SET P022 P006
SFTON3D P022
SMOVL C00031 BC00031 V=166.7  +MOVJ EC00031
MOVL C00032 BC00032 V=1000.0  +MOVJ EC00032 VJ=100.00
'EndPath S4094
MOVJ C00033 BC00033 VJ=100.00  +MOVJ EC00033 VJ=100.00
'Path S4205
SFTOF3D
MOVJ C00034 BC00034 VJ=100.00  +MOVJ EC00034 VJ=100.00
MOVL C00035 BC00035 V=666.7  +MOVJ EC00035 VJ=100.00
SMOVL C00036 BC00036 V=166.7  +MOVJ EC00036
SREFP 3 C00037 BC00037  +REFP EC00037
CALL JOB:SEARCH-R1-S13D
SET P050 P006
SFTON3D P050
SMOVL C00038 BC00038 V=166.7  +MOVJ EC00038
SREFP 3 C00039 BC00039  +REFP EC00039
CALL JOB:SEARCH-R1-S13D
SET P050 P006
SFTON3D P050
SMOVL C00040 BC00040 V=166.7  +MOVJ EC00040
SMOVL C00041 BC00041 V=250.0  +MOVJ EC00041
SMOVL C00042 BC00042 V=166.7  +MOVJ EC00042
SREFP 3 C00043 BC00043  +REFP EC00043
CALL JOB:SEARCH-R1-S13D
SET P050 P006
SFTON3D P050
SMOVL C00044 BC00044 V=250.0  +MOVJ EC00044
'EndPath S4205
'Path S4206
SFTOF3D
MOVL C00045 BC00045 V=1000.0  +MOVJ EC00045 VJ=100.00
SMOVL C00046 BC00046 V=166.7  +MOVJ EC00046
SREFP 3 C00047 BC00047  +REFP EC00047
CALL JOB:SEARCH-R1-S13D
SET P051 P006
SFTON3D P051
SMOVL C00048 BC00048 V=166.7  +MOVJ EC00048
SREFP 3 C00049 BC00049  +REFP EC00049
CALL JOB:SEARCH-R1-S13D
SET P051 P006
SFTON3D P051
SMOVL C00050 BC00050 V=166.7  +MOVJ EC00050
SMOVL C00051 BC00051 V=250.0  +MOVJ EC00051
SREFP 3 C00052 BC00052  +REFP EC00052
CALL JOB:SEARCH-R1-S13D
SET P051 P006
SFTON3D P051
SMOVL C00053 BC00053 V=250.0  +MOVJ EC00053
MOVL C00054 BC00054 V=1000.0  +MOVJ EC00054 VJ=100.00
'EndPath S4206
MOVJ C00055 BC00055 VJ=100.00  +MOVJ EC00055 VJ=100.00
'Path S4207
SFTOF3D
MOVJ C00056 BC00056 VJ=100.00  +MOVJ EC00056 VJ=100.00
MOVL C00057 BC00057 V=666.7  +MOVJ EC00057 VJ=100.00
SMOVL C00058 BC00058 V=166.7  +MOVJ EC00058
SREFP 3 C00059 BC00059  +REFP EC00059
CALL JOB:SEARCH-R1-S13D
SET P054 P006
SFTON3D P054
SMOVL C00060 BC00060 V=250.0  +MOVJ EC00060
SMOVL C00061 BC00061 V=233.3  +MOVJ EC00061
SMOVL C00062 BC00062 V=166.7  +MOVJ EC00062
SREFP 3 C00063 BC00063  +REFP EC00063
CALL JOB:SEARCH-R1-S13D
SET P054 P006
SFTON3D P054
SMOVL C00064 BC00064 V=166.7  +MOVJ EC00064
SMOVL C00065 BC00065 V=416.7  +MOVJ EC00065
SMOVL C00066 BC00066 V=250.0  +MOVJ EC00066
SREFP 3 C00067 BC00067  +REFP EC00067
CALL JOB:SEARCH-R1-S13D
SET P054 P006
SFTON3D P054
SMOVL C00068 BC00068 V=250.0  +MOVJ EC00068
MOVL C00069 BC00069 V=1000.0  +MOVJ EC00069 VJ=100.00
'EndPath S4207
'Path S4095
SFTOF3D
MOVJ C00070 BC00070 VJ=100.00  +MOVJ EC00070 VJ=100.00
MOVJ C00071 BC00071 VJ=100.00  +MOVJ EC00071 VJ=100.00
SMOVL C00072 BC00072 V=200.0  +MOVJ EC00072
SREFP 3 C00073 BC00073  +REFP EC00073
CALL JOB:SEARCH-R1-S13D
SET P089 P006
SFTON3D P089
SMOVL C00074 BC00074 V=166.7  +MOVJ EC00074
SMOVL C00075 BC00075 V=166.7  +MOVJ EC00075
SREFP 3 C00076 BC00076  +REFP EC00076
CALL JOB:SEARCH-R1-S13D
SET P089 P006
SFTON3D P089
SMOVL C00077 BC00077 V=166.7  +MOVJ EC00077
SMOVL C00078 BC00078 V=166.7  +MOVJ EC00078
SREFP 3 C00079 BC00079  +REFP EC00079
CALL JOB:SEARCH-R1-S13D
SET P089 P006
SFTON3D P089
SMOVL C00080 BC00080 V=166.7  +MOVJ EC00080
SMOVL C00081 BC00081 V=1000.0  +MOVJ EC00081
SFTOF3D
MOVJ C00082 BC00082 VJ=100.00  +MOVJ EC00082 VJ=100.00
MOVL C00083 BC00083 V=666.7  +MOVJ EC00083 VJ=100.00
SMOVL C00084 BC00084 V=166.7  +MOVJ EC00084
SREFP 3 C00085 BC00085  +REFP EC00085
CALL JOB:SEARCH-R1-S13D
SET P034 P006
SFTON3D P034
SMOVL C00086 BC00086 V=250.0  +MOVJ EC00086
SMOVL C00087 BC00087 V=233.3  +MOVJ EC00087
SMOVL C00088 BC00088 V=166.7  +MOVJ EC00088
SREFP 3 C00089 BC00089  +REFP EC00089
CALL JOB:SEARCH-R1-S13D
SET P034 P006
SFTON3D P034
SMOVL C00090 BC00090 V=166.7  +MOVJ EC00090
SMOVL C00091 BC00091 V=166.7  +MOVJ EC00091
SREFP 3 C00092 BC00092  +REFP EC00092
CALL JOB:SEARCH-R1-S13D
SET P034 P006
SFTON3D P034
SMOVL C00093 BC00093 V=166.7  +MOVJ EC00093
MOVJ C00094 BC00094 VJ=50.00  +MOVJ EC00094 VJ=30.00
'EndPath S4095
'Path S4096
SFTOF3D
MOVJ C00095 BC00095 VJ=50.00  +MOVJ EC00095 VJ=30.00
MOVJ C00096 BC00096 VJ=50.00  +MOVJ EC00096 VJ=30.00
MOVJ C00097 BC00097 VJ=50.00  +MOVJ EC00097 VJ=30.00
SMOVL C00098 BC00098 V=166.7  +MOVJ EC00098
SREFP 3 C00099 BC00099  +REFP EC00099
CALL JOB:SEARCH-R1-S13D
SET P061 P006
SFTON3D P061
SMOVL C00100 BC00100 V=166.7  +MOVJ EC00100
SREFP 3 C00101 BC00101  +REFP EC00101
CALL JOB:SEARCH-R1-S13D
SET P061 P006
SFTON3D P061
SMOVL C00102 BC00102 V=166.7  +MOVJ EC00102
SFTOF3D
SMOVL C00103 BC00103 V=666.7  +MOVJ EC00103
SMOVL C00104 BC00104 V=166.7  +MOVJ EC00104
SREFP 3 C00105 BC00105  +REFP EC00105
CALL JOB:SEARCH-R1-S13D
SET P062 P006
SFTON3D P062
SMOVL C00106 BC00106 V=166.7  +MOVJ EC00106
SREFP 3 C00107 BC00107  +REFP EC00107
CALL JOB:SEARCH-R1-S13D
SET P062 P006
SFTON3D P062
SMOVL C00108 BC00108 V=250.0  +MOVJ EC00108
SFTOF3D
SMOVL C00109 BC00109 V=500.0  +MOVJ EC00109
SMOVL C00110 BC00110 V=166.7  +MOVJ EC00110
SREFP 3 C00111 BC00111  +REFP EC00111
CALL JOB:SEARCH-R1-S13D
SET P063 P006
SFTON3D P063
SMOVL C00112 BC00112 V=166.7  +MOVJ EC00112
SREFP 3 C00113 BC00113  +REFP EC00113
CALL JOB:SEARCH-R1-S13D
SET P063 P006
SFTON3D P063
SMOVL C00114 BC00114 V=166.7  +MOVJ EC00114
SFTOF3D
SMOVL C00115 BC00115 V=1000.0  +MOVJ EC00115
MOVJ C00116 BC00116 VJ=100.00  +MOVJ EC00116 VJ=30.00
MOVJ C00117 BC00117 VJ=50.00  +MOVJ EC00117 VJ=30.00
MOVJ C00118 BC00118 VJ=100.00  +MOVJ EC00118 VJ=100.00
MOVL C00119 BC00119 V=666.7  +MOVJ EC00119 VJ=100.00
SMOVL C00120 BC00120 V=166.7  +MOVJ EC00120
SREFP 3 C00121 BC00121  +REFP EC00121
CALL JOB:SEARCH-R1-S13D
SET P023 P006
SFTON3D P023
SMOVL C00122 BC00122 V=166.7  +MOVJ EC00122
SMOVL C00123 BC00123 V=333.3  +MOVJ EC00123
SMOVL C00124 BC00124 V=166.7  +MOVJ EC00124
SREFP 3 C00125 BC00125  +REFP EC00125
CALL JOB:SEARCH-R1-S13D
SET P023 P006
SFTON3D P023
SMOVL C00126 BC00126 V=166.7  +MOVJ EC00126
SMOVL C00127 BC00127 V=166.7  +MOVJ EC00127
SREFP 3 C00128 BC00128  +REFP EC00128
CALL JOB:SEARCH-R1-S13D
SET P023 P006
SFTON3D P023
SMOVL C00129 BC00129 V=166.7  +MOVJ EC00129
MOVL C00130 BC00130 V=1000.0  +MOVJ EC00130 VJ=100.00
'EndPath S4096
MOVJ C00131 BC00131 VJ=100.00  +MOVJ EC00131 VJ=100.00
'Path S4097
SFTOF3D
MOVJ C00132 BC00132 VJ=100.00  +MOVJ EC00132 VJ=100.00
MOVL C00133 BC00133 V=666.7  +MOVJ EC00133 VJ=100.00
SMOVL C00134 BC00134 V=166.7  +MOVJ EC00134
SREFP 3 C00135 BC00135  +REFP EC00135
CALL JOB:SEARCH-R1-S13D
SET P024 P006
SFTON3D P024
SMOVL C00136 BC00136 V=166.7  +MOVJ EC00136
SREFP 3 C00137 BC00137  +REFP EC00137
CALL JOB:SEARCH-R1-S13D
SET P024 P006
SFTON3D P024
SMOVL C00138 BC00138 V=166.7  +MOVJ EC00138
SMOVL C00139 BC00139 V=166.7  +MOVJ EC00139
SREFP 3 C00140 BC00140  +REFP EC00140
CALL JOB:SEARCH-R1-S13D
SET P024 P006
SFTON3D P024
SMOVL C00141 BC00141 V=166.7  +MOVJ EC00141
MOVL C00142 BC00142 V=1000.0  +MOVJ EC00142 VJ=100.00
'EndPath S4097
'Path S4098
SFTOF3D
MOVJ C00143 BC00143 VJ=100.00  +MOVJ EC00143 VJ=100.00
MOVL C00144 BC00144 V=666.7  +MOVJ EC00144 VJ=100.00
SMOVL C00145 BC00145 V=166.7  +MOVJ EC00145
SREFP 3 C00146 BC00146  +REFP EC00146
CALL JOB:SEARCH-R1-S13D
SET P035 P006
SFTON3D P035
SMOVL C00147 BC00147 V=166.7  +MOVJ EC00147
SREFP 3 C00148 BC00148  +REFP EC00148
CALL JOB:SEARCH-R1-S13D
SET P035 P006
SFTON3D P035
SMOVL C00149 BC00149 V=166.7  +MOVJ EC00149
SMOVL C00150 BC00150 V=166.7  +MOVJ EC00150
SMOVL C00151 BC00151 V=166.7  +MOVJ EC00151
SREFP 3 C00152 BC00152  +REFP EC00152
CALL JOB:SEARCH-R1-S13D
SET P035 P006
SFTON3D P035
SMOVL C00153 BC00153 V=166.7  +MOVJ EC00153
MOVL C00154 BC00154 V=1000.0  +MOVJ EC00154 VJ=100.00
'EndPath S4098
'Path S4099
SFTOF3D
MOVJ C00155 BC00155 VJ=100.00  +MOVJ EC00155 VJ=100.00
MOVL C00156 BC00156 V=666.7  +MOVJ EC00156 VJ=100.00
SMOVL C00157 BC00157 V=166.7  +MOVJ EC00157
SREFP 3 C00158 BC00158  +REFP EC00158
CALL JOB:SEARCH-R1-S13D
SET P029 P006
SFTON3D P029
SMOVL C00159 BC00159 V=166.7  +MOVJ EC00159
SREFP 3 C00160 BC00160  +REFP EC00160
CALL JOB:SEARCH-R1-S13D
SET P029 P006
SFTON3D P029
SMOVL C00161 BC00161 V=166.7  +MOVJ EC00161
SMOVL C00162 BC00162 V=250.0  +MOVJ EC00162
SMOVL C00163 BC00163 V=166.7  +MOVJ EC00163
SREFP 3 C00164 BC00164  +REFP EC00164
CALL JOB:SEARCH-R1-S13D
SET P029 P006
SFTON3D P029
SMOVL C00165 BC00165 V=166.7  +MOVJ EC00165
'EndPath S4099
'Path S4855
SFTOF3D
MOVL C00166 BC00166 V=666.7  +MOVJ EC00166 VJ=100.00
SMOVL C00167 BC00167 V=166.7  +MOVJ EC00167
SREFP 3 C00168 BC00168  +REFP EC00168
CALL JOB:SEARCH-R1-S13D
SET P071 P006
SFTON3D P071
SMOVL C00169 BC00169 V=166.7  +MOVJ EC00169
SREFP 3 C00170 BC00170  +REFP EC00170
CALL JOB:SEARCH-R1-S13D
SET P071 P006
SFTON3D P071
SMOVL C00171 BC00171 V=166.7  +MOVJ EC00171
SMOVL C00172 BC00172 V=166.7  +MOVJ EC00172
SREFP 3 C00173 BC00173  +REFP EC00173
CALL JOB:SEARCH-R1-S13D
SET P071 P006
SFTON3D P071
SMOVL C00174 BC00174 V=166.7  +MOVJ EC00174
MOVL C00175 BC00175 V=1000.0  +MOVJ EC00175 VJ=100.00
'EndPath S4855
'Path S4856
SFTOF3D
MOVJ C00176 BC00176 VJ=100.00  +MOVJ EC00176 VJ=100.00
MOVL C00177 BC00177 V=666.7  +MOVJ EC00177 VJ=100.00
SMOVL C00178 BC00178 V=166.7  +MOVJ EC00178
SREFP 3 C00179 BC00179  +REFP EC00179
CALL JOB:SEARCH-R1-S13D
SET P072 P006
SFTON3D P072
SMOVL C00180 BC00180 V=166.7  +MOVJ EC00180
SREFP 3 C00181 BC00181  +REFP EC00181
CALL JOB:SEARCH-R1-S13D
SET P072 P006
SFTON3D P072
SMOVL C00182 BC00182 V=166.7  +MOVJ EC00182
MOVL C00183 BC00183 V=1000.0  +MOVJ EC00183 VJ=100.00
'EndPath S4856
MOVJ C00184 BC00184 VJ=100.00  +MOVJ EC00184 VJ=100.00
'Path S4857
SFTOF3D
MOVJ C00185 BC00185 VJ=100.00  +MOVJ EC00185 VJ=100.00
MOVL C00186 BC00186 V=666.7  +MOVJ EC00186 VJ=100.00
SMOVL C00187 BC00187 V=166.7  +MOVJ EC00187
SREFP 3 C00188 BC00188  +REFP EC00188
CALL JOB:SEARCH-R1-S13D
SET P073 P006
SFTON3D P073
SMOVL C00189 BC00189 V=166.7  +MOVJ EC00189
SMOVL C00190 BC00190 V=166.7  +MOVJ EC00190
SREFP 3 C00191 BC00191  +REFP EC00191
CALL JOB:SEARCH-R1-S13D
SET P073 P006
SFTON3D P073
SMOVL C00192 BC00192 V=166.7  +MOVJ EC00192
SMOVL C00193 BC00193 V=166.7  +MOVJ EC00193
SREFP 3 C00194 BC00194  +REFP EC00194
CALL JOB:SEARCH-R1-S13D
SET P073 P006
SFTON3D P073
SMOVL C00195 BC00195 V=166.7  +MOVJ EC00195
MOVL C00196 BC00196 V=1000.0  +MOVJ EC00196 VJ=100.00
'EndPath S4857
MOVJ C00197 BC00197 VJ=100.00  +MOVJ EC00197 VJ=100.00
'Path S4858
SFTOF3D
MOVJ C00198 BC00198 VJ=100.00  +MOVJ EC00198 VJ=100.00
MOVL C00199 BC00199 V=666.7  +MOVJ EC00199 VJ=100.00
SMOVL C00200 BC00200 V=166.7  +MOVJ EC00200
SREFP 3 C00201 BC00201  +REFP EC00201
CALL JOB:SEARCH-R1-S13D
SET P074 P006
SFTON3D P074
SMOVL C00202 BC00202 V=166.7  +MOVJ EC00202
SREFP 3 C00203 BC00203  +REFP EC00203
CALL JOB:SEARCH-R1-S13D
SET P074 P006
SFTON3D P074
SMOVL C00204 BC00204 V=166.7  +MOVJ EC00204
MOVL C00205 BC00205 V=1000.0  +MOVJ EC00205 VJ=100.00
'EndPath S4858
MOVJ C00206 BC00206 VJ=100.00  +MOVJ EC00206 VJ=100.00
MOVJ C00207 BC00207 VJ=100.00  +MOVJ EC00207 VJ=100.00
'Path S4100
SFTOF3D
MOVJ C00208 BC00208 VJ=100.00  +MOVJ EC00208 VJ=100.00
MOVL C00209 BC00209 V=666.7  +MOVJ EC00209 VJ=100.00
SMOVL C00210 BC00210 V=166.7  +MOVJ EC00210
SREFP 3 C00211 BC00211  +REFP EC00211
CALL JOB:SEARCH-R1-S13D
SET P026 P006
SFTON3D P026
SMOVL C00212 BC00212 V=166.7  +MOVJ EC00212
SREFP 3 C00213 BC00213  +REFP EC00213
CALL JOB:SEARCH-R1-S13D
SET P026 P006
SFTON3D P026
SMOVL C00214 BC00214 V=166.7  +MOVJ EC00214
SMOVL C00215 BC00215 V=666.7  +MOVJ EC00215
SMOVL C00216 BC00216 V=666.7  +MOVJ EC00216
SMOVL C00217 BC00217 V=666.7  +MOVJ EC00217
SMOVL C00218 BC00218 V=166.7  +MOVJ EC00218
SREFP 3 C00219 BC00219  +REFP EC00219
CALL JOB:SEARCH-R1-S13D
SET P026 P006
SFTON3D P026
SMOVL C00220 BC00220 V=250.0  +MOVJ EC00220
SMOVL C00221 BC00221 V=666.7  +MOVJ EC00221
MOVL C00222 BC00222 V=1000.0  +MOVJ EC00222 VJ=100.00
'EndPath S4100
MOVJ C00223 BC00223 VJ=50.00  +MOVJ EC00223 VJ=100.00
'Path S4101
SFTOF3D
MOVJ C00224 BC00224 VJ=50.00  +MOVJ EC00224 VJ=100.00
MOVL C00225 BC00225 V=666.7  +MOVJ EC00225 VJ=100.00
SMOVL C00226 BC00226 V=166.7  +MOVJ EC00226
SREFP 3 C00227 BC00227  +REFP EC00227
CALL JOB:SEARCH-R1-S13D
SET P025 P006
SFTON3D P025
SMOVL C00228 BC00228 V=166.7  +MOVJ EC00228
SREFP 3 C00229 BC00229  +REFP EC00229
CALL JOB:SEARCH-R1-S13D
SET P025 P006
SFTON3D P025
SMOVL C00230 BC00230 V=166.7  +MOVJ EC00230
SMOVL C00231 BC00231 V=333.3  +MOVJ EC00231
SMOVL C00232 BC00232 V=166.7  +MOVJ EC00232
SREFP 3 C00233 BC00233  +REFP EC00233
CALL JOB:SEARCH-R1-S13D
SET P025 P006
SFTON3D P025
SMOVL C00234 BC00234 V=166.7  +MOVJ EC00234
MOVL C00235 BC00235 V=1000.0  +MOVJ EC00235 VJ=100.00
'EndPath S4101
MOVJ C00236 BC00236 VJ=100.00  +MOVJ EC00236 VJ=100.00
'Path S4102
SFTOF3D
MOVJ C00237 BC00237 VJ=100.00  +MOVJ EC00237 VJ=100.00
MOVL C00238 BC00238 V=666.7  +MOVJ EC00238 VJ=100.00
SMOVL C00239 BC00239 V=166.7  +MOVJ EC00239
SREFP 3 C00240 BC00240  +REFP EC00240
CALL JOB:SEARCH-R1-S13D
SET P028 P006
SFTON3D P028
SMOVL C00241 BC00241 V=166.7  +MOVJ EC00241
SREFP 3 C00242 BC00242  +REFP EC00242
CALL JOB:SEARCH-R1-S13D
SET P028 P006
SFTON3D P028
SMOVL C00243 BC00243 V=166.7  +MOVJ EC00243
SMOVL C00244 BC00244 V=333.3  +MOVJ EC00244
SMOVL C00245 BC00245 V=166.7  +MOVJ EC00245
SREFP 3 C00246 BC00246  +REFP EC00246
CALL JOB:SEARCH-R1-S13D
SET P028 P006
SFTON3D P028
SMOVL C00247 BC00247 V=166.7  +MOVJ EC00247
MOVL C00248 BC00248 V=1000.0  +MOVJ EC00248 VJ=100.00
'EndPath S4102
MOVJ C00249 BC00249 VJ=100.00  +MOVJ EC00249 VJ=100.00
'Path S4103
SFTOF3D
MOVJ C00250 BC00250 VJ=100.00  +MOVJ EC00250 VJ=100.00
MOVL C00251 BC00251 V=666.7  +MOVJ EC00251 VJ=100.00
SMOVL C00252 BC00252 V=166.7  +MOVJ EC00252
SREFP 3 C00253 BC00253  +REFP EC00253
CALL JOB:SEARCH-R1-S13D
SET P033 P006
SFTON3D P033
SMOVL C00254 BC00254 V=166.7  +MOVJ EC00254
SMOVL C00255 BC00255 V=166.7  +MOVJ EC00255
SREFP 3 C00256 BC00256  +REFP EC00256
CALL JOB:SEARCH-R1-S13D
SET P033 P006
SFTON3D P033
SMOVL C00257 BC00257 V=166.7  +MOVJ EC00257
SMOVL C00258 BC00258 V=166.7  +MOVJ EC00258
SMOVL C00259 BC00259 V=166.7  +MOVJ EC00259
SREFP 3 C00260 BC00260  +REFP EC00260
CALL JOB:SEARCH-R1-S13D
SET P033 P006
SFTON3D P033
SMOVL C00261 BC00261 V=166.7  +MOVJ EC00261
MOVL C00262 BC00262 V=1000.0  +MOVJ EC00262 VJ=100.00
'EndPath S4103
'Path S4104
SFTOF3D
MOVJ C00263 BC00263 VJ=100.00  +MOVJ EC00263 VJ=100.00
MOVL C00264 BC00264 V=666.7  +MOVJ EC00264 VJ=100.00
SMOVL C00265 BC00265 V=166.7  +MOVJ EC00265
SREFP 3 C00266 BC00266  +REFP EC00266
CALL JOB:SEARCH-R1-S13D
SET P027 P006
SFTON3D P027
SMOVL C00267 BC00267 V=250.0  +MOVJ EC00267
SMOVL C00268 BC00268 V=166.7  +MOVJ EC00268
SREFP 3 C00269 BC00269  +REFP EC00269
CALL JOB:SEARCH-R1-S13D
SET P027 P006
SFTON3D P027
SMOVL C00270 BC00270 V=166.7  +MOVJ EC00270
SMOVL C00271 BC00271 V=166.7  +MOVJ EC00271
SREFP 3 C00272 BC00272  +REFP EC00272
CALL JOB:SEARCH-R1-S13D
SET P027 P006
SFTON3D P027
SMOVL C00273 BC00273 V=166.7  +MOVJ EC00273
MOVL C00274 BC00274 V=1000.0  +MOVJ EC00274 VJ=100.00
'EndPath S4104
MOVJ C00275 BC00275 VJ=100.00  +MOVJ EC00275 VJ=100.00
'Path S4105
SFTOF3D
MOVJ C00276 BC00276 VJ=100.00  +MOVJ EC00276 VJ=100.00
MOVL C00277 BC00277 V=666.7  +MOVJ EC00277 VJ=100.00
SMOVL C00278 BC00278 V=166.7  +MOVJ EC00278
SREFP 3 C00279 BC00279  +REFP EC00279
CALL JOB:SEARCH-R1-S13D
SET P030 P006
SFTON3D P030
SMOVL C00280 BC00280 V=166.7  +MOVJ EC00280
SREFP 3 C00281 BC00281  +REFP EC00281
CALL JOB:SEARCH-R1-S13D
SET P030 P006
SFTON3D P030
SMOVL C00282 BC00282 V=166.7  +MOVJ EC00282
MOVL C00283 BC00283 V=1000.0  +MOVJ EC00283 VJ=100.00
'EndPath S4105
'Path S4106
SFTOF3D
MOVJ C00284 BC00284 VJ=100.00  +MOVJ EC00284 VJ=100.00
MOVL C00285 BC00285 V=666.7  +MOVJ EC00285 VJ=100.00
SMOVL C00286 BC00286 V=166.7  +MOVJ EC00286
SREFP 3 C00287 BC00287  +REFP EC00287
CALL JOB:SEARCH-R1-S13D
SET P031 P006
SFTON3D P031
SMOVL C00288 BC00288 V=166.7  +MOVJ EC00288
SREFP 3 C00289 BC00289  +REFP EC00289
CALL JOB:SEARCH-R1-S13D
SET P031 P006
SFTON3D P031
SMOVL C00290 BC00290 V=166.7  +MOVJ EC00290
MOVL C00291 BC00291 V=1000.0  +MOVJ EC00291 VJ=100.00
'EndPath S4106
MOVJ C00292 BC00292 VJ=100.00  +MOVJ EC00292 VJ=100.00
'Path S4107
SFTOF3D
MOVJ C00293 BC00293 VJ=100.00  +MOVJ EC00293 VJ=100.00
MOVL C00294 BC00294 V=666.7  +MOVJ EC00294 VJ=100.00
SMOVL C00295 BC00295 V=166.7  +MOVJ EC00295
SREFP 3 C00296 BC00296  +REFP EC00296
CALL JOB:SEARCH-R1-S13D
SET P032 P006
SFTON3D P032
SMOVL C00297 BC00297 V=166.7  +MOVJ EC00297
SREFP 3 C00298 BC00298  +REFP EC00298
CALL JOB:SEARCH-R1-S13D
SET P032 P006
SFTON3D P032
SMOVL C00299 BC00299 V=166.7  +MOVJ EC00299
SMOVL C00300 BC00300 V=250.0  +MOVJ EC00300
SMOVL C00301 BC00301 V=166.7  +MOVJ EC00301
SREFP 3 C00302 BC00302  +REFP EC00302
CALL JOB:SEARCH-R1-S13D
SET P032 P006
SFTON3D P032
SMOVL C00303 BC00303 V=166.7  +MOVJ EC00303
MOVL C00304 BC00304 V=1000.0  +MOVJ EC00304 VJ=100.00
'EndPath S4107
'
MOVJ C00305 BC00305 VJ=100.00  +MOVJ EC00305 VJ=100.00
'Path S4208
SFTOF3D
MOVJ C00306 BC00306 VJ=100.00  +MOVJ EC00306 VJ=100.00
MOVL C00307 BC00307 V=666.7  +MOVJ EC00307 VJ=100.00
SMOVL C00308 BC00308 V=166.7  +MOVJ EC00308
SREFP 3 C00309 BC00309  +REFP EC00309
CALL JOB:SEARCH-R1-S13D
SET P052 P006
SFTON3D P052
SMOVL C00310 BC00310 V=166.7  +MOVJ EC00310
SREFP 3 C00311 BC00311  +REFP EC00311
CALL JOB:SEARCH-R1-S13D
SET P052 P006
SFTON3D P052
SMOVL C00312 BC00312 V=166.7  +MOVJ EC00312
SFTOF3D
MOVL C00313 BC00313 V=1000.0  +MOVJ EC00313 VJ=100.00
SMOVL C00314 BC00314 V=500.0  +MOVJ EC00314
SMOVL C00315 BC00315 V=166.7  +MOVJ EC00315
SREFP 3 C00316 BC00316  +REFP EC00316
CALL JOB:SEARCH-R1-S13D
SET P088 P006
SFTON3D P088
SMOVL C00317 BC00317 V=166.7  +MOVJ EC00317
SMOVL C00318 BC00318 V=166.7  +MOVJ EC00318
SMOVL C00319 BC00319 V=166.7  +MOVJ EC00319
SREFP 3 C00320 BC00320  +REFP EC00320
CALL JOB:SEARCH-R1-S13D
SET P088 P006
SFTON3D P088
SMOVL C00321 BC00321 V=333.3  +MOVJ EC00321
SMOVL C00322 BC00322 V=666.7  +MOVJ EC00322
SFTOF3D
'EndPath S4208
MOVJ C00323 BC00323 VJ=100.00  +MOVJ EC00323 VJ=100.00
'Path S4209
SFTOF3D
MOVJ C00324 BC00324 VJ=100.00  +MOVJ EC00324 VJ=100.00
MOVL C00325 BC00325 V=666.7  +MOVJ EC00325 VJ=100.00
SMOVL C00326 BC00326 V=166.7  +MOVJ EC00326
SREFP 3 C00327 BC00327  +REFP EC00327
CALL JOB:SEARCH-R1-S13D
SET P053 P006
SFTON3D P053
SMOVL C00328 BC00328 V=166.7  +MOVJ EC00328
SMOVL C00329 BC00329 V=166.7  +MOVJ EC00329
SREFP 3 C00330 BC00330  +REFP EC00330
CALL JOB:SEARCH-R1-S13D
SET P053 P006
SFTON3D P053
SMOVL C00331 BC00331 V=166.7  +MOVJ EC00331
MOVL C00332 BC00332 V=1000.0  +MOVJ EC00332 VJ=100.00
'EndPath S4209
*BP1
MOVJ C00333 BC00333 VJ=100.00  +MOVJ EC00333 VJ=100.00
'Path W4108
SFTOF3D
SFTON3D P033
MOVJ C00334 BC00334 VJ=100.00  +MOVJ EC00334 VJ=100.00
SMOVL C00335 BC00335 V=666.7  +MOVJ EC00335
SMOVL C00336 BC00336 V=166.7 PL=0  +MOVJ EC00336
MACRO1 MJ#(0) ARGF14
ARCON
SMOVL C00337 BC00337 V=9.2  +MOVJ EC00337
ARCOF
SMOVL C00338 BC00338 V=800.0  +MOVJ EC00338
SMOVL C00339 BC00339 V=1000.0  +MOVJ EC00339
SFTOF3D
'EndPath W4108
'Path W4109
SFTOF3D
MOVJ C00340 BC00340 VJ=100.00  +MOVJ EC00340 VJ=100.00
MOVJ C00341 BC00341 VJ=100.00  +MOVJ EC00341 VJ=100.00
'Path W4110
SFTOF3D
SFTON3D P033
MOVJ C00342 BC00342 VJ=100.00  +MOVJ EC00342 VJ=100.00
SMOVL C00343 BC00343 V=800.0  +MOVJ EC00343
SMOVL C00344 BC00344 V=133.3 PL=0  +MOVJ EC00344
MACRO1 MJ#(0) ARGF9
ARCON
SMOVL C00345 BC00345 V=11.7  +MOVJ EC00345
SMOVL C00346 BC00346 V=11.7  +MOVJ EC00346
SMOVL C00347 BC00347 V=11.7  +MOVJ EC00347
ARCOF
SMOVL C00348 BC00348 V=800.0  +MOVJ EC00348
SMOVL C00349 BC00349 V=1000.0  +MOVJ EC00349
SFTOF3D
'EndPath W4110
MOVJ C00350 BC00350 VJ=100.00  +MOVJ EC00350 VJ=100.00
'9
MOVJ C00351 BC00351 VJ=100.00  +MOVJ EC00351 VJ=100.00
'Path W4111
SFTOF3D
SFTON3D P026
MOVJ C00352 BC00352 VJ=100.00  +MOVJ EC00352 VJ=100.00
SMOVL C00353 BC00353 V=666.7  +MOVJ EC00353
SMOVL C00354 BC00354 V=166.7 PL=0  +MOVJ EC00354
MACRO1 MJ#(0) ARGF14
ARCON
SMOVL C00355 BC00355 V=9.2  +MOVJ EC00355
ARCOF
SMOVL C00356 BC00356 V=800.0  +MOVJ EC00356
SMOVL C00357 BC00357 V=1000.0  +MOVJ EC00357
SFTOF3D
'EndPath W4111
'Path W4112
SFTOF3D
SFTON3D P026
MOVJ C00358 BC00358 VJ=100.00  +MOVJ EC00358 VJ=100.00
SMOVL C00359 BC00359 V=800.0  +MOVJ EC00359
SMOVL C00360 BC00360 V=150.0 PL=0  +MOVJ EC00360
ARCON
SMOVL C00361 BC00361 V=11.7  +MOVJ EC00361
SMOVL C00362 BC00362 V=11.7  +MOVJ EC00362
SMOVL C00363 BC00363 V=11.7  +MOVJ EC00363
ARCOF
SMOVL C00364 BC00364 V=800.0  +MOVJ EC00364
SMOVL C00365 BC00365 V=1000.0  +MOVJ EC00365
SFTOF3D
MOVJ C00366 BC00366 VJ=100.00  +MOVJ EC00366 VJ=100.00
MOVJ C00367 BC00367 VJ=100.00  +MOVJ EC00367 VJ=100.00
'uwaga na podajnik
'Path W4114
SFTOF3D
SFTON3D P026
MOVJ C00368 BC00368 VJ=100.00  +MOVJ EC00368 VJ=100.00
SMOVL C00369 BC00369 V=800.0  +MOVJ EC00369
SMOVL C00370 BC00370 V=150.0 PL=0  +MOVJ EC00370
ARCON
SMOVL C00371 BC00371 V=11.7  +MOVJ EC00371
SMOVL C00372 BC00372 V=11.7  +MOVJ EC00372
ARCOF
SMOVL C00373 BC00373 V=800.0  +MOVJ EC00373
SMOVL C00374 BC00374 V=1000.0  +MOVJ EC00374
SFTOF3D
'EndPath W4114
'brak dostepu offset drutu 1cm
'Path W4115
SFTOF3D
SFTON3D P026
MOVJ C00375 BC00375 VJ=100.00  +MOVJ EC00375 VJ=100.00
SMOVL C00376 BC00376 V=800.0  +MOVJ EC00376
SMOVL C00377 BC00377 V=150.0 PL=0  +MOVJ EC00377
ARCON
SMOVL C00378 BC00378 V=11.7  +MOVJ EC00378
ARCOF
SMOVL C00379 BC00379 V=800.0  +MOVJ EC00379
SMOVL C00380 BC00380 V=1000.0  +MOVJ EC00380
SFTOF3D
'EndPath W4115
MOVJ C00381 BC00381 VJ=100.00  +MOVJ EC00381 VJ=100.00
'10
'11
MOVJ C00382 BC00382 VJ=100.00  +MOVJ EC00382 VJ=100.00
'Path W4118
SFTOF3D
SFTON3D P025
MOVJ C00383 BC00383 VJ=100.00  +MOVJ EC00383 VJ=100.00
SMOVL C00384 BC00384 V=800.0  +MOVJ EC00384
SMOVL C00385 BC00385 V=166.7  +MOVJ EC00385
ARCON
SMOVL C00386 BC00386 V=9.2  +MOVJ EC00386
SMOVL C00387 BC00387 V=9.2  +MOVJ EC00387
SMOVL C00388 BC00388 V=9.2  +MOVJ EC00388
SMOVL C00389 BC00389 V=9.2  +MOVJ EC00389
SMOVL C00390 BC00390 V=9.2  +MOVJ EC00390
ARCOF
SMOVL C00391 BC00391 V=800.0  +MOVJ EC00391
SMOVL C00392 BC00392 V=1000.0  +MOVJ EC00392
SFTOF3D
'EndPath W4118
'brak dostepu offset drutu 1cm
MOVJ C00393 BC00393 VJ=100.00  +MOVJ EC00393 VJ=100.00
'Path W4117
SFTOF3D
SFTON3D P025
MOVJ C00394 BC00394 VJ=100.00  +MOVJ EC00394 VJ=100.00
SMOVL C00395 BC00395 V=800.0  +MOVJ EC00395
SMOVL C00396 BC00396 V=166.7 PL=0  +MOVJ EC00396
ARCON
SMOVL C00397 BC00397 V=10.0  +MOVJ EC00397
ARCOF
SMOVL C00398 BC00398 V=800.0  +MOVJ EC00398
SMOVL C00399 BC00399 V=1000.0  +MOVJ EC00399
SFTOF3D
'EndPath W4117
'12
MOVJ C00400 BC00400 VJ=100.00  +MOVJ EC00400 VJ=100.00
MOVJ C00401 BC00401 VJ=100.00  +MOVJ EC00401 VJ=100.00
'Path W4859
SFTOF3D
SFTON3D P073
MOVJ C00402 BC00402 VJ=100.00  +MOVJ EC00402 VJ=100.00
SMOVL C00403 BC00403 V=800.0  +MOVJ EC00403
SMOVL C00404 BC00404 V=150.0 PL=0  +MOVJ EC00404
ARCON
SMOVL C00405 BC00405 V=8.3  +MOVJ EC00405
SFTON3D P074
SMOVL C00406 BC00406 V=9.2  +MOVJ EC00406
SMOVL C00407 BC00407 V=9.2  +MOVJ EC00407
ARCOF
SMOVL C00408 BC00408 V=800.0  +MOVJ EC00408
SMOVL C00409 BC00409 V=1000.0  +MOVJ EC00409
SFTOF3D
'EndPath W4859
MOVJ C00410 BC00410 VJ=100.00  +MOVJ EC00410 VJ=100.00
MOVJ C00411 BC00411 VJ=100.00  +MOVJ EC00411 VJ=100.00
'Path W4119
SFTOF3D
SFTON3D P034
MOVJ C00412 BC00412 VJ=100.00  +MOVJ EC00412 VJ=100.00
SMOVL C00413 BC00413 V=800.0  +MOVJ EC00413
SMOVL C00414 BC00414 V=150.0 PL=0  +MOVJ EC00414
ARCON
SMOVL C00415 BC00415 V=10.0  +MOVJ EC00415
SMOVL C00416 BC00416 V=10.0  +MOVJ EC00416
SMOVL C00417 BC00417 V=10.0  +MOVJ EC00417
ARCOF
SMOVL C00418 BC00418 V=800.0  +MOVJ EC00418
SMOVL C00419 BC00419 V=1000.0  +MOVJ EC00419
SFTOF3D
'EndPath W4119
'Path W4210
SFTOF3D
SFTON3D P050
MOVJ C00420 BC00420 VJ=100.00  +MOVJ EC00420 VJ=100.00
SMOVL C00421 BC00421 V=800.0  +MOVJ EC00421
SMOVL C00422 BC00422 V=150.0 PL=0  +MOVJ EC00422
ARCON
SMOVL C00423 BC00423 V=11.7  +MOVJ EC00423
ARCOF
SMOVL C00424 BC00424 V=800.0  +MOVJ EC00424
SMOVL C00425 BC00425 V=1000.0  +MOVJ EC00425
SFTOF3D
'EndPath W4210
'Path W4211
SFTOF3D
SFTON3D P034
MOVJ C00426 BC00426 VJ=100.00  +MOVJ EC00426 VJ=100.00
SMOVL C00427 BC00427 V=800.0  +MOVJ EC00427
SMOVL C00428 BC00428 V=166.7 PL=0  +MOVJ EC00428
ARCON
SWVON WEV#(66)
SMOVL C00429 BC00429 V=9.2  +MOVJ EC00429
SMOVL C00430 BC00430 V=9.2  +MOVJ EC00430
SMOVL C00431 BC00431 V=9.2  +MOVJ EC00431
ARCOF
WVOF
SMOVL C00432 BC00432 V=800.0  +MOVJ EC00432
SMOVL C00433 BC00433 V=1000.0  +MOVJ EC00433
MOVJ C00434 BC00434 VJ=30.00  +MOVJ EC00434 VJ=30.00
MOVJ C00435 BC00435 VJ=30.00  +MOVJ EC00435 VJ=30.00
SFTOF3D
MACRO1 MJ#(0) ARGF6
MOVJ C00436 BC00436 VJ=30.00  +MOVJ EC00436 VJ=30.00
SFTON3D P063
SMOVL C00437 BC00437 V=133.3  +MOVJ EC00437
ARCON
SMOVL C00438 BC00438 V=11.7  +MOVJ EC00438
SMOVL C00439 BC00439 V=11.7  +MOVJ EC00439
SMOVL C00440 BC00440 V=11.7  +MOVJ EC00440
SFTON3D P062
SMOVL C00441 BC00441 V=11.7  +MOVJ EC00441
SMOVL C00442 BC00442 V=11.7  +MOVJ EC00442
SFTON3D P061
SMOVL C00443 BC00443 V=11.0  +MOVJ EC00443
SMOVL C00444 BC00444 V=11.0  +MOVJ EC00444
ARCOF
SMOVL C00445 BC00445 V=250.0  +MOVJ EC00445
SFTOF3D
MOVJ C00446 BC00446 VJ=20.00  +MOVJ EC00446 VJ=20.00
MOVJ C00447 BC00447 VJ=20.00  +MOVJ EC00447 VJ=20.00
MOVJ C00448 BC00448 VJ=30.00  +MOVJ EC00448 VJ=30.00
'EndPath W4211
'Path W4210
SFTOF3D
SFTON3D P054
MOVJ C00449 BC00449 VJ=100.00  +MOVJ EC00449 VJ=100.00
SMOVL C00450 BC00450 V=800.0  +MOVJ EC00450
SMOVL C00451 BC00451 V=150.0 PL=0  +MOVJ EC00451
MACRO1 MJ#(0) ARGF14
ARCON
SWVON WEV#(67)
SMOVL C00452 BC00452 V=10.0  +MOVJ EC00452
SMOVL C00453 BC00453 V=10.0  +MOVJ EC00453
ARCOF
SWVOF
SMOVL C00454 BC00454 V=800.0  +MOVJ EC00454
SMOVL C00455 BC00455 V=1000.0  +MOVJ EC00455
SFTOF3D
'EndPath W4210
'Path W4121
SFTOF3D
SFTON3D P028
MOVJ C00456 BC00456 VJ=100.00  +MOVJ EC00456 VJ=100.00
SMOVL C00457 BC00457 V=800.0  +MOVJ EC00457
SMOVL C00458 BC00458 V=150.0 PL=0  +MOVJ EC00458
ARCON
SMOVL C00459 BC00459 V=9.2  +MOVJ EC00459
SMOVL C00460 BC00460 V=9.2  +MOVJ EC00460
SMOVL C00461 BC00461 V=9.2  +MOVJ EC00461
ARCOF
SMOVL C00462 BC00462 V=800.0  +MOVJ EC00462
SMOVL C00463 BC00463 V=1000.0  +MOVJ EC00463
SFTOF3D
'EndPath W4121
'brak dostepu offset 5mm
MOVJ C00464 BC00464 VJ=100.00  +MOVJ EC00464 VJ=100.00
'Path W4122
SFTOF3D
SFTON3D P028
MOVJ C00465 BC00465 VJ=100.00  +MOVJ EC00465 VJ=100.00
SMOVL C00466 BC00466 V=800.0  +MOVJ EC00466
SMOVL C00467 BC00467 V=166.7 PL=0  +MOVJ EC00467
ARCON
SMOVL C00468 BC00468 V=11.7  +MOVJ EC00468
ARCOF
SMOVL C00469 BC00469 V=800.0  +MOVJ EC00469
SMOVL C00470 BC00470 V=1000.0  +MOVJ EC00470
SFTOF3D
'EndPath W4122
MOVJ C00471 BC00471 VJ=100.00  +MOVJ EC00471 VJ=100.00
'13
MOVJ C00472 BC00472 VJ=100.00  +MOVJ EC00472 VJ=100.00
'Path W4123
SFTOF3D
SFTON3D P030
MOVJ C00473 BC00473 VJ=100.00  +MOVJ EC00473 VJ=100.00
SMOVL C00474 BC00474 V=800.0  +MOVJ EC00474
SMOVL C00475 BC00475 V=150.0 PL=0  +MOVJ EC00475
MACRO1 MJ#(0) ARGF9
ARCON
SWVON WEV#(10)
SFTON3D P031
SMOVL C00476 BC00476 V=12.5  +MOVJ EC00476
ARCOF
SWVOF
SMOVL C00477 BC00477 V=800.0  +MOVJ EC00477
SMOVL C00478 BC00478 V=1000.0  +MOVJ EC00478
SFTOF3D
'EndPath W4123
'14
'15-brak
'Path W4212
SFTOF3D
SFTON3D P052
MOVJ C00479 BC00479 VJ=100.00  +MOVJ EC00479 VJ=100.00
SMOVL C00480 BC00480 V=800.0  +MOVJ EC00480
SMOVL C00481 BC00481 V=150.0 PL=0  +MOVJ EC00481
ARCON
SMOVL C00482 BC00482 V=10.8  +MOVJ EC00482
SMOVL C00483 BC00483 V=10.8  +MOVJ EC00483
SMOVL C00484 BC00484 V=10.8  +MOVJ EC00484
ARCOF
SMOVL C00485 BC00485 V=800.0  +MOVJ EC00485
MACRO1 MJ#(0) ARGF6
SMOVL C00486 BC00486 V=333.3  +MOVJ EC00486
SFTOF3D
'DODAC SHIFT
SFTON3D P088
SMOVL C00487 BC00487 V=133.3  +MOVJ EC00487
ARCON
SMOVL C00488 BC00488 V=10.8  +MOVJ EC00488
ARCOF
SMOVL C00489 BC00489 V=250.0  +MOVJ EC00489
SMOVL C00490 BC00490 V=1000.0  +MOVJ EC00490
SFTOF3D
'EndPath W4212
'16
'Path W4213
SFTOF3D
SFTON3D P053
MOVJ C00491 BC00491 VJ=100.00  +MOVJ EC00491 VJ=100.00
SMOVL C00492 BC00492 V=800.0  +MOVJ EC00492
SMOVL C00493 BC00493 V=150.0 PL=0  +MOVJ EC00493
MACRO1 MJ#(0) ARGF9
ARCON
SMOVL C00494 BC00494 V=10.8  +MOVJ EC00494
SMOVL C00495 BC00495 V=10.8  +MOVJ EC00495
SMOVL C00496 BC00496 V=10.8  +MOVJ EC00496
ARCOF
SMOVL C00497 BC00497 V=800.0  +MOVJ EC00497
SMOVL C00498 BC00498 V=1000.0  +MOVJ EC00498
SFTOF3D
'EndPath W4213
'Path W4124
SFTOF3D
SFTON3D P029
MOVJ C00499 BC00499 VJ=100.00  +MOVJ EC00499 VJ=100.00
SMOVL C00500 BC00500 V=800.0  +MOVJ EC00500
SMOVL C00501 BC00501 V=166.7 PL=0  +MOVJ EC00501
MACRO1 MJ#(0) ARGF14
ARCON
SMOVL C00502 BC00502 V=10.0  +MOVJ EC00502
SMOVL C00503 BC00503 V=10.0  +MOVJ EC00503
ARCOF
SMOVL C00504 BC00504 V=800.0  +MOVJ EC00504
SMOVL C00505 BC00505 V=1000.0  +MOVJ EC00505
SFTOF3D
'EndPath W4124
MOVJ C00506 BC00506 VJ=100.00  +MOVJ EC00506 VJ=100.00
'Path W4125
SFTOF3D
SFTON3D P029
MOVJ C00507 BC00507 VJ=100.00  +MOVJ EC00507 VJ=100.00
SMOVL C00508 BC00508 V=800.0  +MOVJ EC00508
SMOVL C00509 BC00509 V=150.0 PL=0  +MOVJ EC00509
ARCON
SMOVL C00510 BC00510 V=11.7  +MOVJ EC00510
SMOVL C00511 BC00511 V=11.7  +MOVJ EC00511
SMOVL C00512 BC00512 V=11.7  +MOVJ EC00512
ARCOF
SMOVL C00513 BC00513 V=800.0  +MOVJ EC00513
SMOVL C00514 BC00514 V=1000.0  +MOVJ EC00514
SFTOF3D
'EndPath W4125
MOVJ C00515 BC00515 VJ=100.00  +MOVJ EC00515 VJ=100.00
'Path W4126
SFTOF3D
SFTON3D P029
MOVJ C00516 BC00516 VJ=100.00  +MOVJ EC00516 VJ=100.00
SMOVL C00517 BC00517 V=800.0  +MOVJ EC00517
SMOVL C00518 BC00518 V=166.7 PL=0  +MOVJ EC00518
ARCON
SMOVL C00519 BC00519 V=11.7  +MOVJ EC00519
ARCON
SMOVL C00520 BC00520 V=11.7  +MOVJ EC00520
SMOVL C00521 BC00521 V=11.7  +MOVJ EC00521
ARCOF
SMOVL C00522 BC00522 V=800.0  +MOVJ EC00522
SMOVL C00523 BC00523 V=1000.0  +MOVJ EC00523
SFTOF3D
'EndPath W4126
MOVJ C00524 BC00524 VJ=100.00  +MOVJ EC00524 VJ=100.00
'17
'Path W4127
SFTOF3D
SFTON3D P027
MOVJ C00525 BC00525 VJ=100.00  +MOVJ EC00525 VJ=100.00
SMOVL C00526 BC00526 V=800.0  +MOVJ EC00526
SMOVL C00527 BC00527 V=150.0 PL=0  +MOVJ EC00527
ARCON
SMOVL C00528 BC00528 V=10.0  +MOVJ EC00528
ARCOF
SMOVL C00529 BC00529 V=800.0  +MOVJ EC00529
SMOVL C00530 BC00530 V=1000.0  +MOVJ EC00530
SFTOF3D
'EndPath W4127
'Path W4128
SFTOF3D
SFTON3D P027
MOVJ C00531 BC00531 VJ=100.00  +MOVJ EC00531 VJ=100.00
SMOVL C00532 BC00532 V=800.0  +MOVJ EC00532
SMOVL C00533 BC00533 V=150.0 PL=0  +MOVJ EC00533
ARCON
SMOVL C00534 BC00534 V=11.7  +MOVJ EC00534
ARCOF
SMOVL C00535 BC00535 V=800.0  +MOVJ EC00535
SMOVL C00536 BC00536 V=1000.0  +MOVJ EC00536
SFTOF3D
'EndPath W4128
'Path W4129
SFTOF3D
SFTON3D P027
MOVJ C00537 BC00537 VJ=100.00  +MOVJ EC00537 VJ=100.00
SMOVL C00538 BC00538 V=800.0  +MOVJ EC00538
SMOVL C00539 BC00539 V=150.0 PL=0  +MOVJ EC00539
SMOVL C00540 BC00540 V=16.7  +MOVJ EC00540
ARCOF
SMOVL C00541 BC00541 V=800.0  +MOVJ EC00541
SMOVL C00542 BC00542 V=1000.0  +MOVJ EC00542
SFTOF3D
'EndPath W4129
'18
MOVJ C00543 BC00543 VJ=100.00  +MOVJ EC00543 VJ=100.00
'Path W4130
SFTOF3D
SFTON3D P024
MOVJ C00544 BC00544 VJ=100.00  +MOVJ EC00544 VJ=100.00
SMOVL C00545 BC00545 V=800.0  +MOVJ EC00545
SMOVL C00546 BC00546 V=150.0 PL=0  +MOVJ EC00546
ARCON
SMOVL C00547 BC00547 V=9.2  +MOVJ EC00547
SMOVL C00548 BC00548 V=9.2  +MOVJ EC00548
SMOVL C00549 BC00549 V=9.2  +MOVJ EC00549
SMOVL C00550 BC00550 V=9.2  +MOVJ EC00550
ARCOF
SMOVL C00551 BC00551 V=800.0  +MOVJ EC00551
SMOVL C00552 BC00552 V=1000.0  +MOVJ EC00552
SFTOF3D
'EndPath W4130
'Path W4860
SFTOF3D
SFTON3D P071
MOVJ C00553 BC00553 VJ=100.00  +MOVJ EC00553 VJ=100.00
SMOVL C00554 BC00554 V=800.0  +MOVJ EC00554
SMOVL C00555 BC00555 V=150.0 PL=0  +MOVJ EC00555
MACRO1 MJ#(0) ARGF9
ARCON
SMOVL C00556 BC00556 V=9.2  +MOVJ EC00556
SFTON3D P072
ARCON
SMOVL C00557 BC00557 V=9.2  +MOVJ EC00557
SMOVL C00558 BC00558 V=9.2  +MOVJ EC00558
ARCOF
SMOVL C00559 BC00559 V=800.0  +MOVJ EC00559
SMOVL C00560 BC00560 V=1000.0  +MOVJ EC00560
SFTOF3D
'EndPath W4860
'19
MOVJ C00561 BC00561 VJ=100.00  +MOVJ EC00561 VJ=100.00
'Path W4131
SFTOF3D
SFTON3D P023
MOVJ C00562 BC00562 VJ=100.00  +MOVJ EC00562 VJ=100.00
SMOVL C00563 BC00563 V=800.0  +MOVJ EC00563
SMOVL C00564 BC00564 V=166.7 PL=0  +MOVJ EC00564
MACRO1 MJ#(0) ARGF9
ARCON
SWVON WEV#(60)
SMOVL C00565 BC00565 V=7.5  +MOVJ EC00565
SMOVL C00566 BC00566 V=7.5  +MOVJ EC00566
SMOVL C00567 BC00567 V=7.5  +MOVJ EC00567
ARCOF
SWVOF
SMOVL C00568 BC00568 V=800.0  +MOVJ EC00568
SMOVL C00569 BC00569 V=1000.0  +MOVJ EC00569
SFTOF3D
'EndPath W4131
MOVJ C00570 BC00570 VJ=100.00  +MOVJ EC00570 VJ=100.00
'Path W4214
SFTOF3D
SFTON3D P089
MOVJ C00571 BC00571 VJ=100.00  +MOVJ EC00571 VJ=100.00
SMOVL C00572 BC00572 V=800.0  +MOVJ EC00572
SMOVL C00573 BC00573 V=150.0 PL=0  +MOVJ EC00573
MACRO1 MJ#(0) ARGF9
ARCON
SMOVL C00574 BC00574 V=9.2  +MOVJ EC00574
SFTON3D P050
SMOVL C00575 BC00575 V=9.2  +MOVJ EC00575
SMOVL C00576 BC00576 V=9.2  +MOVJ EC00576
ARCOF
SMOVL C00577 BC00577 V=800.0  +MOVJ EC00577
SMOVL C00578 BC00578 V=1000.0  +MOVJ EC00578
SFTOF3D
'EndPath W4214
'Path W4215
SFTOF3D
SFTON3D P051
MOVJ C00579 BC00579 VJ=100.00  +MOVJ EC00579 VJ=100.00
SMOVL C00580 BC00580 V=800.0  +MOVJ EC00580
SMOVL C00581 BC00581 V=150.0 PL=0  +MOVJ EC00581
MACRO1 MJ#(0) ARGF9
ARCON
SWVON WEV#(60)
SMOVL C00582 BC00582 V=7.5  +MOVJ EC00582
SMOVL C00583 BC00583 V=7.5  +MOVJ EC00583
SMOVL C00584 BC00584 V=7.5  +MOVJ EC00584
ARCOF
SWVOF
SMOVL C00585 BC00585 V=800.0  +MOVJ EC00585
SMOVL C00586 BC00586 V=1000.0  +MOVJ EC00586
SFTOF3D
'EndPath W4215
MOVJ C00587 BC00587 VJ=100.00  +MOVJ EC00587 VJ=100.00
'20
'offset 5mm
MOVJ C00588 BC00588 VJ=100.00  +MOVJ EC00588 VJ=100.00
MOVJ C00589 BC00589 VJ=100.00  +MOVJ EC00589 VJ=100.00
'Path W4132
SFTOF3D
SFTON3D P032
MOVJ C00590 BC00590 VJ=100.00  +MOVJ EC00590 VJ=100.00
SMOVL C00591 BC00591 V=800.0  +MOVJ EC00591
SMOVL C00592 BC00592 V=150.0 PL=0  +MOVJ EC00592
ARCON
SMOVL C00593 BC00593 V=10.0  +MOVJ EC00593
SMOVL C00594 BC00594 V=10.0  +MOVJ EC00594
ARCOF
SMOVL C00595 BC00595 V=800.0  +MOVJ EC00595
SMOVL C00596 BC00596 V=1000.0  +MOVJ EC00596
SFTOF3D
JUMP *FFF
'EndPath W4132
'Path W4133
SFTOF3D
SFTON3D P032
MOVJ C00597 BC00597 VJ=100.00  +MOVJ EC00597 VJ=100.00
SMOVL C00598 BC00598 V=800.0  +MOVJ EC00598
SMOVL C00599 BC00599 V=166.7 PL=0  +MOVJ EC00599
ARCON
SMOVL C00600 BC00600 V=10.0  +MOVJ EC00600
ARCOF
SMOVL C00601 BC00601 V=800.0  +MOVJ EC00601
SMOVL C00602 BC00602 V=1000.0  +MOVJ EC00602
SFTOF3D
'EndPath W4133
'Path W4134
SFTOF3D
SFTON3D P032
MOVJ C00603 BC00603 VJ=100.00  +MOVJ EC00603 VJ=100.00
SMOVL C00604 BC00604 V=800.0  +MOVJ EC00604
SMOVL C00605 BC00605 V=150.0 PL=0  +MOVJ EC00605
ARCON
SMOVL C00606 BC00606 V=10.0  +MOVJ EC00606
ARCOF
SMOVL C00607 BC00607 V=800.0  +MOVJ EC00607
*FFF
SMOVL C00608 BC00608 V=1000.0  +MOVJ EC00608
SFTOF3D
'EndPath W4134
'offset 5mm
MOVJ C00609 BC00609 VJ=100.00  +MOVJ EC00609 VJ=100.00
'Path W4135
SFTOF3D
SFTON3D P032
MOVJ C00610 BC00610 VJ=100.00  +MOVJ EC00610 VJ=100.00
SMOVL C00611 BC00611 V=800.0  +MOVJ EC00611
SMOVL C00612 BC00612 V=166.7 PL=0  +MOVJ EC00612
ARCON
SMOVL C00613 BC00613 V=10.0  +MOVJ EC00613
ARCOF
SMOVL C00614 BC00614 V=800.0  +MOVJ EC00614
SMOVL C00615 BC00615 V=1000.0  +MOVJ EC00615
SFTOF3D
'EndPath W4135
MOVJ C00616 BC00616 VJ=100.00  +MOVJ EC00616 VJ=100.00
'Path W4136
SFTOF3D
SFTON3D P032
MOVJ C00617 BC00617 VJ=100.00  +MOVJ EC00617 VJ=100.00
SMOVL C00618 BC00618 V=800.0  +MOVJ EC00618
SMOVL C00619 BC00619 V=166.7 PL=0  +MOVJ EC00619
ARCON
SMOVL C00620 BC00620 V=11.7  +MOVJ EC00620
SMOVL C00621 BC00621 V=11.7  +MOVJ EC00621
ARCOF
SMOVL C00622 BC00622 V=800.0  +MOVJ EC00622
SMOVL C00623 BC00623 V=1000.0  +MOVJ EC00623
SFTOF3D
'EndPath W4136
MOVJ C00624 BC00624 VJ=100.00  +MOVJ EC00624 VJ=100.00
MOVJ C00625 BC00625 VJ=100.00  +MOVJ EC00625 VJ=100.00
'Path W4137
SFTOF3D
SFTON3D P021
MOVJ C00626 BC00626 VJ=100.00  +MOVJ EC00626 VJ=100.00
SMOVL C00627 BC00627 V=800.0  +MOVJ EC00627
SMOVL C00628 BC00628 V=150.0 PL=0  +MOVJ EC00628
MACRO1 MJ#(0) ARGF9
ARCON
SFTON3D P022
SMOVL C00629 BC00629 V=10.0  +MOVJ EC00629
ARCOF
SMOVL C00630 BC00630 V=800.0  +MOVJ EC00630
SMOVL C00631 BC00631 V=1000.0  +MOVJ EC00631
SFTOF3D
'EndPath W4137
MOVJ C00632 BC00632 VJ=100.00  +MOVJ EC00632 VJ=100.00
'Path W4724
SFTOF3D
SFTON3D P095
MOVJ C00633 BC00633 VJ=100.00  +MOVJ EC00633 VJ=100.00
SMOVL C00634 BC00634 V=800.0  +MOVJ EC00634
SMOVL C00635 BC00635 V=150.0 PL=0  +MOVJ EC00635
ARCON
SMOVL C00636 BC00636 V=10.0  +MOVJ EC00636
SMOVL C00637 BC00637 V=10.0  +MOVJ EC00637
SMOVL C00638 BC00638 V=10.0  +MOVJ EC00638
ARCOF
SMOVL C00639 BC00639 V=800.0  +MOVJ EC00639
SMOVL C00640 BC00640 V=1000.0  +MOVJ EC00640
SFTOF3D
'EndPath W4724
'Path W4725
SFTOF3D
SFTON3D P096
MOVJ C00641 BC00641 VJ=100.00  +MOVJ EC00641 VJ=100.00
SMOVL C00642 BC00642 V=800.0  +MOVJ EC00642
SMOVL C00643 BC00643 V=150.0 PL=0  +MOVJ EC00643
ARCON
SMOVL C00644 BC00644 V=10.0  +MOVJ EC00644
SMOVL C00645 BC00645 V=10.0  +MOVJ EC00645
ARCOF
SMOVL C00646 BC00646 V=800.0  +MOVJ EC00646
SMOVL C00647 BC00647 V=1000.0  +MOVJ EC00647
SFTOF3D
'EndPath W4725
MOVJ C00648 BC00648 VJ=100.00  +MOVJ EC00648 VJ=100.00
'Path W4861
SFTOF3D
SFTON3D P071
MOVJ C00649 BC00649 VJ=100.00  +MOVJ EC00649 VJ=100.00
SMOVL C00650 BC00650 V=800.0  +MOVJ EC00650
SMOVL C00651 BC00651 V=150.0 PL=0  +MOVJ EC00651
MACRO1 MJ#(0) ARGF14
ARCON
SMOVL C00652 BC00652 V=9.2  +MOVJ EC00652
SFTON3D P073
SMOVL C00653 BC00653 V=9.2  +MOVJ EC00653
SMOVL C00654 BC00654 V=9.2  +MOVJ EC00654
ARCOF
SMOVL C00655 BC00655 V=800.0  +MOVJ EC00655
SMOVL C00656 BC00656 V=1000.0  +MOVJ EC00656
SFTOF3D
'EndPath W4861
MOVJ C00657 BC00657 VJ=100.00  +MOVJ EC00657 VJ=100.00
MOVJ C00658 BC00658 VJ=100.00  +MOVJ EC00658 VJ=100.00
CALL JOB:CLEAN-R1_KM_NEW
'cut_wire_dol
'cut_wire_dol
'cut_wire_dol
MOVJ C00659 BC00659 VJ=100.00  +MOVJ EC00659 VJ=100.00
MOVJ C00660 BC00660 VJ=100.00  +MOVJ EC00660 VJ=100.00
MOVJ C00661 BC00661 VJ=100.00  +MOVJ EC00661 VJ=100.00
'Path S4138
SFTOF3D
MOVJ C00662 BC00662 VJ=100.00  +MOVJ EC00662 VJ=100.00
MOVL C00663 BC00663 V=800.0  +MOVJ EC00663 VJ=100.00
SMOVL C00664 BC00664 V=166.7  +MOVJ EC00664
SREFP 3 C00665 BC00665  +REFP EC00665
CALL JOB:SEARCH-R1-S13D
SET P049 P006
SFTON3D P049
SMOVL C00666 BC00666 V=166.7  +MOVJ EC00666
SMOVL C00667 BC00667 V=100.0  +MOVJ EC00667
SMOVL C00668 BC00668 V=166.7  +MOVJ EC00668
SREFP 3 C00669 BC00669  +REFP EC00669
CALL JOB:SEARCH-R1-S13D
SET P049 P006
SFTON3D P049
SMOVL C00670 BC00670 V=166.7  +MOVJ EC00670
SMOVL C00671 BC00671 V=166.7  +MOVJ EC00671
SMOVL C00672 BC00672 V=166.7  +MOVJ EC00672
SREFP 3 C00673 BC00673  +REFP EC00673
CALL JOB:SEARCH-R1-S13D
SET P049 P006
SFTON3D P049
SMOVL C00674 BC00674 V=166.7  +MOVJ EC00674
MOVL C00675 BC00675 V=800.0  +MOVJ EC00675 VJ=100.00
MOVL C00676 BC00676 V=1000.0  +MOVJ EC00676 VJ=100.00
'EndPath S4138
'Path S4139
SFTOF3D
MOVJ C00677 BC00677 VJ=100.00  +MOVJ EC00677 VJ=100.00
MOVL C00678 BC00678 V=800.0  +MOVJ EC00678 VJ=100.00
SMOVL C00679 BC00679 V=166.7  +MOVJ EC00679
SREFP 3 C00680 BC00680  +REFP EC00680
CALL JOB:SEARCH-R1-S13D
SET P048 P006
SFTON3D P048
SMOVL C00681 BC00681 V=166.7  +MOVJ EC00681
SMOVL C00682 BC00682 V=166.7  +MOVJ EC00682
SREFP 3 C00683 BC00683  +REFP EC00683
CALL JOB:SEARCH-R1-S13D
SET P048 P006
SFTON3D P048
SMOVL C00684 BC00684 V=166.7  +MOVJ EC00684
MOVL C00685 BC00685 V=800.0  +MOVJ EC00685 VJ=100.00
MOVL C00686 BC00686 V=1000.0  +MOVJ EC00686 VJ=100.00
'EndPath S4139
'Path S4140
SFTOF3D
MOVJ C00687 BC00687 VJ=100.00  +MOVJ EC00687 VJ=100.00
MOVL C00688 BC00688 V=800.0  +MOVJ EC00688 VJ=100.00
SMOVL C00689 BC00689 V=166.7  +MOVJ EC00689
SREFP 3 C00690 BC00690  +REFP EC00690
CALL JOB:SEARCH-R1-S13D
SET P047 P006
SFTON3D P047
SMOVL C00691 BC00691 V=166.7  +MOVJ EC00691
SMOVL C00692 BC00692 V=166.7  +MOVJ EC00692
SMOVL C00693 BC00693 V=166.7  +MOVJ EC00693
SREFP 3 C00694 BC00694  +REFP EC00694
CALL JOB:SEARCH-R1-S13D
SET P047 P006
SFTON3D P047
SMOVL C00695 BC00695 V=166.7  +MOVJ EC00695
MOVL C00696 BC00696 V=800.0  +MOVJ EC00696 VJ=100.00
MOVL C00697 BC00697 V=1000.0  +MOVJ EC00697 VJ=100.00
'EndPath S4140
MOVJ C00698 BC00698 VJ=100.00  +MOVJ EC00698 VJ=100.00
MOVJ C00699 BC00699 VJ=100.00  +MOVJ EC00699 VJ=100.00
MOVJ C00700 BC00700 VJ=100.00  +MOVJ EC00700 VJ=100.00
MOVJ C00701 BC00701 VJ=100.00  +MOVJ EC00701 VJ=100.00
'Path S4141
SFTOF3D
MOVJ C00702 BC00702 VJ=20.00  +MOVJ EC00702 VJ=20.00
MOVJ C00703 BC00703 VJ=100.00  +MOVJ EC00703 VJ=100.00
MOVL C00704 BC00704 V=800.0  +MOVJ EC00704 VJ=100.00
SMOVL C00705 BC00705 V=166.7  +MOVJ EC00705
SREFP 3 C00706 BC00706  +REFP EC00706
CALL JOB:SEARCH-R1-S13D
SET P046 P006
SFTON3D P046
SMOVL C00707 BC00707 V=166.7  +MOVJ EC00707
SMOVL C00708 BC00708 V=166.7  +MOVJ EC00708
SREFP 3 C00709 BC00709  +REFP EC00709
CALL JOB:SEARCH-R1-S13D
SET P046 P006
SFTON3D P046
SMOVL C00710 BC00710 V=166.7  +MOVJ EC00710
MOVL C00711 BC00711 V=1000.0  +MOVJ EC00711 VJ=100.00
'EndPath S4141
'Path S4142
SFTOF3D
MOVJ C00712 BC00712 VJ=100.00  +MOVJ EC00712 VJ=100.00
MOVL C00713 BC00713 V=800.0  +MOVJ EC00713 VJ=100.00
SMOVL C00714 BC00714 V=166.7  +MOVJ EC00714
SREFP 3 C00715 BC00715  +REFP EC00715
CALL JOB:SEARCH-R1-S13D
SET P045 P006
SFTON3D P045
SMOVL C00716 BC00716 V=166.7  +MOVJ EC00716
SMOVL C00717 BC00717 V=166.7  +MOVJ EC00717
SREFP 3 C00718 BC00718  +REFP EC00718
CALL JOB:SEARCH-R1-S13D
SET P045 P006
SFTON3D P045
SMOVL C00719 BC00719 V=166.7  +MOVJ EC00719
MOVL C00720 BC00720 V=1000.0  +MOVJ EC00720 VJ=100.00
'EndPath S4142
'Path S4143
SFTOF3D
MOVJ C00721 BC00721 VJ=100.00  +MOVJ EC00721 VJ=100.00
MOVL C00722 BC00722 V=800.0  +MOVJ EC00722 VJ=100.00
SMOVL C00723 BC00723 V=166.7  +MOVJ EC00723
SREFP 3 C00724 BC00724  +REFP EC00724
CALL JOB:SEARCH-R1-S13D
SET P044 P006
SFTON3D P044
SMOVL C00725 BC00725 V=166.7  +MOVJ EC00725
SMOVL C00726 BC00726 V=166.7  +MOVJ EC00726
SREFP 3 C00727 BC00727  +REFP EC00727
CALL JOB:SEARCH-R1-S13D
SET P044 P006
SFTON3D P044
SMOVL C00728 BC00728 V=166.7  +MOVJ EC00728
MOVL C00729 BC00729 V=1000.0  +MOVJ EC00729 VJ=100.00
'EndPath S4143
MOVJ C00730 BC00730 VJ=100.00  +MOVJ EC00730 VJ=100.00
MOVJ C00731 BC00731 VJ=100.00  +MOVJ EC00731 VJ=100.00
'Path S4144
SFTOF3D
MOVJ C00732 BC00732 VJ=100.00  +MOVJ EC00732 VJ=100.00
MOVL C00733 BC00733 V=800.0  +MOVJ EC00733 VJ=100.00
SMOVL C00734 BC00734 V=166.7  +MOVJ EC00734
SREFP 3 C00735 BC00735  +REFP EC00735
CALL JOB:SEARCH-R1-S13D
SET P043 P006
SFTON3D P043
SMOVL C00736 BC00736 V=166.7  +MOVJ EC00736
SMOVL C00737 BC00737 V=166.7  +MOVJ EC00737
SREFP 3 C00738 BC00738  +REFP EC00738
CALL JOB:SEARCH-R1-S13D
SET P043 P006
SFTON3D P043
SMOVL C00739 BC00739 V=166.7  +MOVJ EC00739
MOVL C00740 BC00740 V=1000.0  +MOVJ EC00740 VJ=100.00
'EndPath S4144
'Path S4145
SFTOF3D
MOVJ C00741 BC00741 VJ=100.00  +MOVJ EC00741 VJ=100.00
MOVL C00742 BC00742 V=800.0  +MOVJ EC00742 VJ=100.00
SMOVL C00743 BC00743 V=166.7  +MOVJ EC00743
SREFP 3 C00744 BC00744  +REFP EC00744
CALL JOB:SEARCH-R1-S13D
SET P042 P006
SFTON3D P042
SMOVL C00745 BC00745 V=166.7  +MOVJ EC00745
SMOVL C00746 BC00746 V=166.7  +MOVJ EC00746
SREFP 3 C00747 BC00747  +REFP EC00747
CALL JOB:SEARCH-R1-S13D
SET P042 P006
SFTON3D P042
SMOVL C00748 BC00748 V=166.7  +MOVJ EC00748
MOVL C00749 BC00749 V=1000.0  +MOVJ EC00749 VJ=100.00
'EndPath S4145
'Path S4146
SFTOF3D
MOVJ C00750 BC00750 VJ=100.00  +MOVJ EC00750 VJ=100.00
MOVL C00751 BC00751 V=666.7  +MOVJ EC00751 VJ=100.00
SMOVL C00752 BC00752 V=166.7  +MOVJ EC00752
SREFP 3 C00753 BC00753  +REFP EC00753
CALL JOB:SEARCH-R1-S13D
SET P041 P006
SFTON3D P041
SMOVL C00754 BC00754 V=250.0  +MOVJ EC00754
SMOVL C00755 BC00755 V=166.7  +MOVJ EC00755
SREFP 3 C00756 BC00756  +REFP EC00756
CALL JOB:SEARCH-R1-S13D
SET P041 P006
SFTON3D P041
SMOVL C00757 BC00757 V=166.7  +MOVJ EC00757
SMOVL C00758 BC00758 V=166.7  +MOVJ EC00758
SREFP 3 C00759 BC00759  +REFP EC00759
CALL JOB:SEARCH-R1-S13D
SET P041 P006
SFTON3D P041
SMOVL C00760 BC00760 V=166.7  +MOVJ EC00760
MOVL C00761 BC00761 V=1000.0  +MOVJ EC00761 VJ=100.00
'EndPath S4146
'Path S4147
SFTOF3D
MOVJ C00762 BC00762 VJ=100.00  +MOVJ EC00762 VJ=100.00
SMOVL C00763 BC00763 V=666.7  +MOVJ EC00763
SMOVL C00764 BC00764 V=166.7  +MOVJ EC00764
SREFP 3 C00765 BC00765  +REFP EC00765
CALL JOB:SEARCH-R1-S13D
SET P040 P006
SFTON3D P040
SMOVL C00766 BC00766 V=166.7  +MOVJ EC00766
SMOVL C00767 BC00767 V=800.0  +MOVJ EC00767
SMOVL C00768 BC00768 V=166.7  +MOVJ EC00768
SREFP 3 C00769 BC00769  +REFP EC00769
CALL JOB:SEARCH-R1-S13D
SET P040 P006
SFTON3D P040
SMOVL C00770 BC00770 V=166.7  +MOVJ EC00770
SMOVL C00771 BC00771 V=166.7  +MOVJ EC00771
SREFP 3 C00772 BC00772  +REFP EC00772
CALL JOB:SEARCH-R1-S13D
SET P040 P006
SFTON3D P040
SMOVL C00773 BC00773 V=166.7  +MOVJ EC00773
MOVL C00774 BC00774 V=1000.0  +MOVJ EC00774 VJ=100.00
'EndPath S4147
'Path W4148
SFTOF3D
SFTON3D P040
MOVJ C00775 BC00775 VJ=100.00  +MOVJ EC00775 VJ=100.00
SMOVL C00776 BC00776 V=800.0  +MOVJ EC00776
SMOVL C00777 BC00777 V=150.0 PL=0  +MOVJ EC00777
ARCON
SMOVL C00778 BC00778 V=10.0  +MOVJ EC00778
ARCOF
SMOVL C00779 BC00779 V=800.0  +MOVJ EC00779
SMOVL C00780 BC00780 V=1000.0  +MOVJ EC00780
SFTOF3D
'EndPath W4148
'Path W4149
SFTOF3D
SFTON3D P040
MOVJ C00781 BC00781 VJ=100.00  +MOVJ EC00781 VJ=100.00
SMOVL C00782 BC00782 V=800.0  +MOVJ EC00782
SMOVL C00783 BC00783 V=150.0 PL=0  +MOVJ EC00783
ARCON
SMOVL C00784 BC00784 V=11.7  +MOVJ EC00784
ARCOF
SMOVL C00785 BC00785 V=800.0  +MOVJ EC00785
SMOVL C00786 BC00786 V=1000.0  +MOVJ EC00786
SFTOF3D
'EndPath W4149
'Path W4150
SFTOF3D
SFTON3D P040
MOVJ C00787 BC00787 VJ=15.00  +MOVJ EC00787 VJ=15.00
MOVJ C00788 BC00788 VJ=100.00  +MOVJ EC00788 VJ=100.00
SMOVL C00789 BC00789 V=800.0  +MOVJ EC00789
SMOVL C00790 BC00790 V=150.0 PL=0  +MOVJ EC00790
ARCON
SMOVL C00791 BC00791 V=11.7  +MOVJ EC00791
ARCOF
SMOVL C00792 BC00792 V=800.0  +MOVJ EC00792
SMOVL C00793 BC00793 V=1000.0  +MOVJ EC00793
SFTOF3D
'EndPath W4150
'
MOVJ C00794 BC00794 VJ=100.00  +MOVJ EC00794 VJ=100.00
MOVJ C00795 BC00795 VJ=100.00  +MOVJ EC00795 VJ=100.00
'Path W4151
SFTOF3D
SFTON3D P045
MOVJ C00796 BC00796 VJ=100.00  +MOVJ EC00796 VJ=100.00
SMOVL C00797 BC00797 V=800.0  +MOVJ EC00797
SMOVL C00798 BC00798 V=150.0 PL=0  +MOVJ EC00798
MACRO1 MJ#(0) ARGF9
ARCON
SMOVL C00799 BC00799 V=11.7  +MOVJ EC00799
ARCOF
SMOVL C00800 BC00800 V=800.0  +MOVJ EC00800
SMOVL C00801 BC00801 V=1000.0  +MOVJ EC00801
SFTOF3D
'EndPath W4151
'Path W4152
SFTOF3D
SFTON3D P044
MOVJ C00802 BC00802 VJ=100.00  +MOVJ EC00802 VJ=100.00
SMOVL C00803 BC00803 V=800.0  +MOVJ EC00803
SMOVL C00804 BC00804 V=166.7 PL=0  +MOVJ EC00804
ARCON
SMOVL C00805 BC00805 V=11.7  +MOVJ EC00805
ARCOF
SMOVL C00806 BC00806 V=800.0  +MOVJ EC00806
SMOVL C00807 BC00807 V=1000.0  +MOVJ EC00807
SFTOF3D
'EndPath W4152
'Path W4153
SFTOF3D
SFTON3D P046
MOVJ C00808 BC00808 VJ=100.00  +MOVJ EC00808 VJ=100.00
SMOVL C00809 BC00809 V=800.0  +MOVJ EC00809
SMOVL C00810 BC00810 V=166.7 PL=0  +MOVJ EC00810
MACRO1 MJ#(0) ARGF14
ARCON
SMOVL C00811 BC00811 V=10.0  +MOVJ EC00811
SMOVL C00812 BC00812 V=10.0  +MOVJ EC00812
ARCOF
SMOVL C00813 BC00813 V=800.0  +MOVJ EC00813
SMOVL C00814 BC00814 V=1000.0  +MOVJ EC00814
SFTOF3D
'EndPath W4153
MOVJ C00815 BC00815 VJ=20.00  +MOVJ EC00815 VJ=20.00
MOVJ C00816 BC00816 VJ=20.00  +MOVJ EC00816 VJ=20.00
MOVJ C00817 BC00817 VJ=100.00  +MOVJ EC00817 VJ=100.00
MOVJ C00818 BC00818 VJ=100.00  +MOVJ EC00818 VJ=100.00
MOVJ C00819 BC00819 VJ=100.00  +MOVJ EC00819 VJ=100.00
MOVJ C00820 BC00820 VJ=100.00  +MOVJ EC00820 VJ=100.00
'1
'uwaga na podajnik
'Path W4154
SFTOF3D
SFTON3D P048
MOVJ C00821 BC00821 VJ=100.00  +MOVJ EC00821 VJ=100.00
SMOVL C00822 BC00822 V=800.0  +MOVJ EC00822
SMOVL C00823 BC00823 V=150.0 PL=0  +MOVJ EC00823
ARCON
SMOVL C00824 BC00824 V=10.0  +MOVJ EC00824
ARCOF
SMOVL C00825 BC00825 V=800.0  +MOVJ EC00825
SMOVL C00826 BC00826 V=1000.0  +MOVJ EC00826
SFTOF3D
'EndPath W4154
'Path W4155
SFTOF3D
SFTON3D P049
MOVJ C00827 BC00827 VJ=100.00  +MOVJ EC00827 VJ=100.00
SMOVL C00828 BC00828 V=800.0  +MOVJ EC00828
SMOVL C00829 BC00829 V=150.0 PL=0  +MOVJ EC00829
MACRO1 MJ#(0) ARGF6
ARCON
SMOVL C00830 BC00830 V=9.2  +MOVJ EC00830
SMOVL C00831 BC00831 V=9.2  +MOVJ EC00831
SMOVL C00832 BC00832 V=9.2  +MOVJ EC00832
SMOVL C00833 BC00833 V=9.2  +MOVJ EC00833
SMOVL C00834 BC00834 V=9.2  +MOVJ EC00834
ARCOF
SMOVL C00835 BC00835 V=800.0  +MOVJ EC00835
MOVJ C00836 BC00836 VJ=20.00  +MOVJ EC00836 VJ=20.00
SMOVL C00837 BC00837 V=166.7  +MOVJ EC00837
ARCON
SMOVL C00838 BC00838 V=10.0  +MOVJ EC00838
ARCOF
SMOVL C00839 BC00839 V=250.0  +MOVJ EC00839
SMOVL C00840 BC00840 V=500.0  +MOVJ EC00840
SMOVL C00841 BC00841 V=500.0  +MOVJ EC00841
SMOVL C00842 BC00842 V=500.0  +MOVJ EC00842
SMOVL C00843 BC00843 V=133.3  +MOVJ EC00843
ARCON
SMOVL C00844 BC00844 V=13.3  +MOVJ EC00844
ARCOF
SMOVL C00845 BC00845 V=166.7  +MOVJ EC00845
SMOVL C00846 BC00846 V=166.7  +MOVJ EC00846
ARCON
SMOVL C00847 BC00847 V=10.0  +MOVJ EC00847
ARCOF
SMOVL C00848 BC00848 V=800.0  +MOVJ EC00848
SFTOF3D
'EndPath W4155
MOVJ C00849 BC00849 VJ=100.00  +MOVJ EC00849 VJ=100.00
MOVJ C00850 BC00850 VJ=100.00  +MOVJ EC00850 VJ=100.00
MOVJ C00851 BC00851 VJ=100.00  +MOVJ EC00851 VJ=100.00
MOVJ C00852 BC00852 VJ=100.00  +MOVJ EC00852 VJ=100.00
MOVJ C00853 BC00853 VJ=20.00  +MOVJ EC00853 VJ=20.00
'2
'Path W4156
SFTOF3D
SFTON3D P043
MOVJ C00854 BC00854 VJ=100.00  +MOVJ EC00854 VJ=100.00
SMOVL C00855 BC00855 V=800.0  +MOVJ EC00855
SMOVL C00856 BC00856 V=166.7 PL=0  +MOVJ EC00856
MACRO1 MJ#(0) ARGF9
ARCON
SMOVL C00857 BC00857 V=11.7  +MOVJ EC00857
ARCOF
SMOVL C00858 BC00858 V=800.0  +MOVJ EC00858
SMOVL C00859 BC00859 V=1000.0  +MOVJ EC00859
SFTOF3D
'EndPath W4156
'Path W4157
SFTOF3D
SFTON3D P042
MOVJ C00860 BC00860 VJ=100.00  +MOVJ EC00860 VJ=100.00
SMOVL C00861 BC00861 V=800.0  +MOVJ EC00861
SMOVL C00862 BC00862 V=150.0 PL=0  +MOVJ EC00862
ARCON
SMOVL C00863 BC00863 V=11.7  +MOVJ EC00863
ARCOF
SMOVL C00864 BC00864 V=800.0  +MOVJ EC00864
SMOVL C00865 BC00865 V=1000.0  +MOVJ EC00865
SFTOF3D
'EndPath W4157
'3
MOVJ C00866 BC00866 VJ=20.00  +MOVJ EC00866 VJ=20.00
MOVJ C00867 BC00867 VJ=100.00  +MOVJ EC00867 VJ=100.00
MOVJ C00868 BC00868 VJ=100.00  +MOVJ EC00868 VJ=100.00
MOVJ C00869 BC00869 VJ=100.00  +MOVJ EC00869 VJ=100.00
MOVJ C00870 BC00870 VJ=100.00  +MOVJ EC00870 VJ=100.00
'Path W4158
SFTOF3D
SFTON3D P047
MOVJ C00871 BC00871 VJ=100.00  +MOVJ EC00871 VJ=100.00
SMOVL C00872 BC00872 V=800.0  +MOVJ EC00872
SMOVL C00873 BC00873 V=150.0 PL=0  +MOVJ EC00873
ARCON
SMOVL C00874 BC00874 V=11.7  +MOVJ EC00874
ARCOF
SMOVL C00875 BC00875 V=800.0  +MOVJ EC00875
SMOVL C00876 BC00876 V=1000.0  +MOVJ EC00876
SFTOF3D
'EndPath W4158
'Path W4159
SFTOF3D
SFTON3D P047
MOVJ C00877 BC00877 VJ=100.00  +MOVJ EC00877 VJ=100.00
SMOVL C00878 BC00878 V=800.0  +MOVJ EC00878
SMOVL C00879 BC00879 V=150.0 PL=0  +MOVJ EC00879
ARCON
SMOVL C00880 BC00880 V=11.7  +MOVJ EC00880
ARCOF
SMOVL C00881 BC00881 V=800.0  +MOVJ EC00881
SMOVL C00882 BC00882 V=1000.0  +MOVJ EC00882
SFTOF3D
'EndPath W4159
MOVJ C00883 BC00883 VJ=100.00  +MOVJ EC00883 VJ=100.00
MOVJ C00884 BC00884 VJ=100.00  +MOVJ EC00884 VJ=100.00
MOVJ C00885 BC00885 VJ=100.00  +MOVJ EC00885 VJ=100.00
MOVJ C00886 BC00886 VJ=100.00  +MOVJ EC00886 VJ=100.00
MOVJ C00887 BC00887 VJ=20.00  +MOVJ EC00887 VJ=20.00
'Path W4160
SFTOF3D
SFTON3D P043
MOVJ C00888 BC00888 VJ=100.00  +MOVJ EC00888 VJ=100.00
SMOVL C00889 BC00889 V=800.0  +MOVJ EC00889
SMOVL C00890 BC00890 V=150.0 PL=0  +MOVJ EC00890
ARCON
SMOVL C00891 BC00891 V=11.7  +MOVJ EC00891
ARCOF
SMOVL C00892 BC00892 V=800.0  +MOVJ EC00892
SMOVL C00893 BC00893 V=1000.0  +MOVJ EC00893
SFTOF3D
'EndPath W4160
'Path W4161
SFTOF3D
SFTON3D P042
MOVJ C00894 BC00894 VJ=100.00  +MOVJ EC00894 VJ=100.00
SMOVL C00895 BC00895 V=800.0  +MOVJ EC00895
SMOVL C00896 BC00896 V=166.7 PL=0  +MOVJ EC00896
ARCON
SMOVL C00897 BC00897 V=11.7  +MOVJ EC00897
ARCOF
SMOVL C00898 BC00898 V=800.0  +MOVJ EC00898
SMOVL C00899 BC00899 V=1000.0  +MOVJ EC00899
SFTOF3D
'EndPath W4161
MOVJ C00900 BC00900 VJ=100.00  +MOVJ EC00900 VJ=100.00
'Path W4162
SFTOF3D
SFTON3D P046
MOVJ C00901 BC00901 VJ=100.00  +MOVJ EC00901 VJ=100.00
SMOVL C00902 BC00902 V=800.0  +MOVJ EC00902
SMOVL C00903 BC00903 V=166.7 PL=0  +MOVJ EC00903
MACRO1 MJ#(0) ARGF14
ARCON
SMOVL C00904 BC00904 V=10.0  +MOVJ EC00904
ARCOF
SMOVL C00905 BC00905 V=800.0  +MOVJ EC00905
SMOVL C00906 BC00906 V=1000.0  +MOVJ EC00906
SFTOF3D
'EndPath W4162
'Path W4163
SFTOF3D
SFTON3D P044
MOVJ C00907 BC00907 VJ=100.00  +MOVJ EC00907 VJ=100.00
SMOVL C00908 BC00908 V=800.0  +MOVJ EC00908
SMOVL C00909 BC00909 V=150.0 PL=0  +MOVJ EC00909
MACRO1 MJ#(0) ARGF9
ARCON
SMOVL C00910 BC00910 V=11.7  +MOVJ EC00910
ARCOF
SMOVL C00911 BC00911 V=800.0  +MOVJ EC00911
SMOVL C00912 BC00912 V=1000.0  +MOVJ EC00912
SFTOF3D
'EndPath W4163
MOVJ C00913 BC00913 VJ=100.00  +MOVJ EC00913 VJ=100.00
'Path W4164
SFTOF3D
SFTON3D P041
MOVJ C00914 BC00914 VJ=100.00  +MOVJ EC00914 VJ=100.00
SMOVL C00915 BC00915 V=800.0  +MOVJ EC00915
SMOVL C00916 BC00916 V=150.0 PL=0  +MOVJ EC00916
MACRO1 MJ#(0) ARGF14
ARCON
SMOVL C00917 BC00917 V=10.0  +MOVJ EC00917
SMOVL C00918 BC00918 V=10.0  +MOVJ EC00918
SMOVL C00919 BC00919 V=10.0  +MOVJ EC00919
ARCOF
SMOVL C00920 BC00920 V=800.0  +MOVJ EC00920
SMOVL C00921 BC00921 V=1000.0  +MOVJ EC00921
SFTOF3D
'EndPath W4164
JUMP *L_1
'Path W4165
SFTOF3D
SFTON3D P041
MOVJ C00922 BC00922 VJ=100.00  +MOVJ EC00922 VJ=100.00
SMOVL C00923 BC00923 V=800.0  +MOVJ EC00923
SMOVL C00924 BC00924 V=150.0 PL=0  +MOVJ EC00924
SMOVL C00925 BC00925 V=10.0  +MOVJ EC00925
ARCOF
SMOVL C00926 BC00926 V=800.0  +MOVJ EC00926
SMOVL C00927 BC00927 V=1000.0  +MOVJ EC00927
SFTOF3D
'EndPath W4165
MOVJ C00928 BC00928 VJ=100.00  +MOVJ EC00928 VJ=100.00
'Path W4166
SFTOF3D
SFTON3D P041
MOVJ C00929 BC00929 VJ=100.00  +MOVJ EC00929 VJ=100.00
SMOVL C00930 BC00930 V=800.0  +MOVJ EC00930
SMOVL C00931 BC00931 V=150.0 PL=0  +MOVJ EC00931
SMOVL C00932 BC00932 V=10.0  +MOVJ EC00932
ARCOF
SMOVL C00933 BC00933 V=800.0  +MOVJ EC00933
SMOVL C00934 BC00934 V=1000.0  +MOVJ EC00934
SFTOF3D
'EndPath W4166
*L_1
MOVJ C00935 BC00935 VJ=100.00  +MOVJ EC00935 VJ=100.00
MOVJ C00936 BC00936 VJ=20.00  +MOVJ EC00936 VJ=20.00
MOVJ C00937 BC00937 VJ=100.00  +MOVJ EC00937 VJ=100.00
MOVJ C00938 BC00938 VJ=100.00  +MOVJ EC00938 VJ=100.00
END
